(*
Nazwa:			P00_PneumaticValves
Opis:			Wyspa pneumatyczna
Wersja:			v1.0
Data:			2025-10-20
Autor:			DP
Urzadzenia:		Obsługa wyspy zaworowej
Konfiguracja:	
Info:
- kazdy zawór to 2 bity
#######################################################
#######################################################
*)



PROGRAM P00_PneumaticValves
VAR
	//ZMIENNE STERUJĄCE WYSPY ZAWOROWEJ
	QABPneumatic641ValveCoils 			AT %Q* 	: ARRAY[1..6] OF BYTE;
	QABPneumatic642ValveCoils 			AT %Q*	: ARRAY[1..5] OF BYTE;
	QABPneumatic643ValveCoils 			AT %Q*	: ARRAY[1..5] OF BYTE;
	QABPneumatic644ValveCoils 			AT %Q*	: ARRAY[1..5] OF BYTE;
	QABPneumatic645ValveCoils 			AT %Q*	: ARRAY[1..2] OF BYTE;
	QABPneumatic646ValveCoils 			AT %Q* 	: ARRAY[1..5] OF BYTE;
	QABPneumatic647ValveCoils 			AT %Q* 	: ARRAY[1..5] OF BYTE;
	QABPneumaticPI641ValveCoils 		AT %Q* 	: ARRAY[1..6] OF BYTE;

	QABPneumatic641PressureRegulator 	AT %Q* 	: ARRAY[1..2] OF BYTE;
	IABPneumatic641PressureRegulator 	AT %I* 	: ARRAY[1..2] OF BYTE;
	QABPneumatic645_1PressureRegulator 	AT %Q* 	: ARRAY[1..2] OF BYTE;
	IABPneumatic645_1PressureRegulator 	AT %I* 	: ARRAY[1..2] OF BYTE;
	QABPneumatic645_2PressureRegulator 	AT %Q* 	: ARRAY[1..2] OF BYTE;
	IABPneumatic645_2PressureRegulator 	AT %I* 	: ARRAY[1..2] OF BYTE;
	
	IABPneumatic641_N11AnalogInput1 	AT %I* 	: ARRAY[1..2] OF BYTE;
	IABPneumatic641_N11AnalogInput2 	AT %I* 	: ARRAY[1..2] OF BYTE;
	IABPneumatic641_N11AnalogInput3 	AT %I* 	: ARRAY[1..2] OF BYTE;
	IABPneumatic641_N11AnalogInput4 	AT %I* 	: ARRAY[1..2] OF BYTE;
	IABPneumatic645_N11AnalogInput1 	AT %I* 	: ARRAY[1..2] OF BYTE;
	IABPneumatic645_N11AnalogInput2 	AT %I* 	: ARRAY[1..2] OF BYTE;
	IABPneumatic645_N11AnalogInput3 	AT %I* 	: ARRAY[1..2] OF BYTE;
	IABPneumatic645_N11AnalogInput4 	AT %I* 	: ARRAY[1..2] OF BYTE;
	                                    
	IABPneumatic641_N12DigitalInput 	AT %I* 	: BYTE;	
	IABPneumatic642_N11DigitalInput 	AT %I* 	: BYTE;	
	IABPneumatic642_N12DigitalInput 	AT %I* 	: BYTE;	
	IABPneumatic642_N13DigitalInput 	AT %I* 	: BYTE;	
	IABPneumatic643_N11DigitalInput 	AT %I* 	: BYTE;	
	IABPneumatic643_N12DigitalInput 	AT %I* 	: BYTE;	
	IABPneumatic643_N13DigitalInput 	AT %I* 	: BYTE;
	IABPneumatic644_N11DigitalInput 	AT %I* 	: BYTE;	
	IABPneumatic644_N12DigitalInput 	AT %I* 	: BYTE;	
	IABPneumatic644_N13DigitalInput 	AT %I* 	: BYTE;
	IABPneumatic645_N12DigitalInput 	AT %I* 	: BYTE;
	IABPneumatic646_N11DigitalInput 	AT %I* 	: BYTE;
	IABPneumatic646_N12DigitalInput 	AT %I* 	: BYTE;
	IABPneumatic646_N13DigitalInput 	AT %I* 	: BYTE;
	IABPneumatic647_N11DigitalInput 	AT %I* 	: BYTE;
	IABPneumatic647_N12DigitalInput 	AT %I* 	: BYTE;
	IABPneumaticPI641_N11DigitalInput 	AT %I* 	: BYTE;
	IABPneumaticPI641_N12DigitalInput 	AT %I* 	: BYTE;
	IABPneumaticPI641_N13DigitalInput 	AT %I* 	: BYTE;
	                                  
	iIABPneumatic645_N11AnalogInput1	:INT;
	iIABPneumatic645_N11AnalogInput2    :INT;
	iIABPneumatic645_N11AnalogInput3    :INT;
	iIABPneumatic645_N11AnalogInput4    :INT;
	iIABPneumatic641_N11AnalogInput1    :INT;
	iIABPneumatic641_N11AnalogInput2    :INT;
	iIABPneumatic641_N11AnalogInput3    :INT;
	iIABPneumatic641_N11AnalogInput4    :INT;
	
	iIABPneumatic641PressureRegulator1				: INT;
	iIABPneumatic641PressureRegulator2				: INT;
	iIABPneumatic645_1PressureRegulator1			: INT;
	iIABPneumatic645_1PressureRegulator2			: INT;
	iIABPneumatic645_2PressureRegulator1			: INT;
	iIABPneumatic645_2PressureRegulator2			: INT;
	
	iQABPneumatic641PressureRegulator1				: INT;
	iQABPneumatic641PressureRegulator2				: INT;	
	iQABPneumatic645_1PressureRegulator1			: INT;
	iQABPneumatic645_1PressureRegulator2			: INT;
	iQABPneumatic645_2PressureRegulator1			: INT;
	iQABPneumatic645_2PressureRegulator2			: INT;	
	                                    
	(*Skalowanie czujników poziomu*)    
	fbiTank1LevelSensorValue 			: FB_4_20mA_TO_INT;
	fbiTank2LevelSensorValue 			: FB_4_20mA_TO_INT;	
	
	lrLidSealerPressureTemp						: LREAL;
	lrGripperScrewerCatchPressureTemp			: LREAL;
	lrGripperScrewerPressureTemp				: LREAL;
	lrDispencercatchPressureTemp				: LREAL;

	
END_VAR

//aVTEM();
//aVTEMSignals();
aAnalogueInput();
aDigitalInput();
aPressureRegulator();
aValveCoil();

ACTION aAnalogueInput:
(*
Nazwa:			aAnalogueInput
Opis:			Zawory pneumatyczne
Wersja:			v0.1
Data:			2024-10-28
Autor:			DP
Urzadzenia:		
Konfiguracja:	
Info:
- Czujnik pozycji Balluff, trzeba skonfigurować na 4-20mA, domyślnie jest na 0-10V
- Instrukcja konfiguracji czujnika: 2s, 1x, 1x (zniknie dioda), 2s (wyjście), 2s (wyjście)
*)

(*************************** 641N1.1 **************************************)
// Wyspa 1 - dozowanie
//AI1 4-20mA 
IABPneumatic641_N11AnalogInput1[1];
IABPneumatic641_N11AnalogInput1[2];
iIABPneumatic641_N11AnalogInput1	:= WORD_TO_INT(F_2Bytes_To_Word(byHigh:=IABPneumatic641_N11AnalogInput1[2],byLow:=IABPneumatic641_N11AnalogInput1[1]));
P02_Dispencers.IbDispencersCatch1SensorValue:=F_Scaling(rValue:=iIABPneumatic641_N11AnalogInput1, 
	rXmin:=		0,		//	0mA
	rXmax:=		32767,	//	23mA
	rYmin:= 	-70000, //	~10000 -> ~10mm (szyjka butelki) zamkniety (chwytak otwiera się na 49mm)
	rYmax:=		135000 );// ~60000 -> ~60mm otwarty
{warning 'dodać błąd czujnika poniżej 4mA i powyżej 20mA'}
IABPneumatic641_N11AnalogInput2[1]; 
IABPneumatic641_N11AnalogInput2[2];
iIABPneumatic641_N11AnalogInput2	:= WORD_TO_INT(F_2Bytes_To_Word(byHigh:=IABPneumatic641_N11AnalogInput2[2],byLow:=IABPneumatic641_N11AnalogInput2[1]));
P02_Dispencers.IbDispencersCatch2SensorValue:=F_Scaling(rValue:=iIABPneumatic641_N11AnalogInput2, 
	rXmin:=		0,		//	0mA
	rXmax:=		32767,	//	23mA
	rYmin:= 	-70000, //	~10000 -> ~10mm (szyjka butelki) zamkniety (chwytak otwiera się na 49mm)
	rYmax:=		135000 );// ~60000 -> ~60mm otwarty

IABPneumatic641_N11AnalogInput3[1]; 
IABPneumatic641_N11AnalogInput3[2]; 
iIABPneumatic641_N11AnalogInput3	:= WORD_TO_INT(F_2Bytes_To_Word(byHigh:=IABPneumatic641_N11AnalogInput3[2],byLow:=IABPneumatic641_N11AnalogInput3[1]));
P02_Dispencers.IbDispencersCatch3SensorValue:=F_Scaling(rValue:=iIABPneumatic641_N11AnalogInput3, 
	rXmin:=		0,		//	0mA
	rXmax:=		32767,	//	23mA
	rYmin:= 	-70000, //	~10000 -> ~10mm (szyjka butelki) zamkniety (chwytak otwiera się na 49mm)
	rYmax:=		135000 );// ~60000 -> ~60mm otwarty

IABPneumatic641_N11AnalogInput4[1]; 	
IABPneumatic641_N11AnalogInput4[2]; 
iIABPneumatic641_N11AnalogInput4	:= WORD_TO_INT(F_2Bytes_To_Word(byHigh:=IABPneumatic641_N11AnalogInput4[2],byLow:=IABPneumatic641_N11AnalogInput4[1]));
P02_Dispencers.IbDispencersCatch4SensorValue:=F_Scaling(rValue:=iIABPneumatic641_N11AnalogInput4, 
	rXmin:=		0,		//	0mA
	rXmax:=		32767,	//	23mA
	rYmin:= 	-70000, //	~10000 -> ~10mm (szyjka butelki) zamkniety (chwytak otwiera się na 49mm)
	rYmax:=		135000 );// ~60000 -> ~60mm otwarty

(*********************Koniec 641N1.1 **************************************)


(*************************** 645N1.1 **************************************)
// Wyspa 5 - zakręcarki i czujnik poziomu
//AI1 4-20mA 
IABPneumatic645_N11AnalogInput1[1];
IABPneumatic645_N11AnalogInput1[2];
iIABPneumatic645_N11AnalogInput1	:= WORD_TO_INT(F_2Bytes_To_Word(byHigh:=IABPneumatic645_N11AnalogInput1[2],byLow:=IABPneumatic645_N11AnalogInput1[1]));
P10_GripperScrewer.IlrGripperScrewer1HeightCV	:=	-0.0023*(iIABPneumatic645_N11AnalogInput1)+52.006 + 2.6788;

IABPneumatic645_N11AnalogInput2[1]; 
IABPneumatic645_N11AnalogInput2[2]; 
iIABPneumatic645_N11AnalogInput2	:= WORD_TO_INT(F_2Bytes_To_Word(byHigh:=IABPneumatic645_N11AnalogInput2[2],byLow:=IABPneumatic645_N11AnalogInput2[1]));
P10_GripperScrewer.IlrGripperScrewer2HeightCV	:=	-0.0023*(iIABPneumatic645_N11AnalogInput2)+52.006 + 2.252;

IABPneumatic645_N11AnalogInput3[1];
IABPneumatic645_N11AnalogInput3[2];
iIABPneumatic645_N11AnalogInput3	:= WORD_TO_INT(F_2Bytes_To_Word(byHigh:=IABPneumatic645_N11AnalogInput3[2],byLow:=IABPneumatic645_N11AnalogInput3[1]));
//iTank1Sensor1Value;//Czujnik poziomu 1
fbiTank1LevelSensorValue(
	iIN:= 	iIABPneumatic645_N11AnalogInput3, 
	rXmin:= 5190,//5513.0, 	// 4mA
	rXmax:= 27307.0, 	// 20mA
	rYmin:= 10.0, 		// 10mm na czujniku to 4mA
	rYmax:= 325.0,		// 325mm na czujniku to 20mA
	bError=>, 			// Bląd <4mA i >20mA
	iOUT=>	VIS.iTank1LevelSensorValue );
fbiTank1LevelSensorValue.bError;

IABPneumatic645_N11AnalogInput4[1];
IABPneumatic645_N11AnalogInput4[2];
iIABPneumatic645_N11AnalogInput4	:= WORD_TO_INT(F_2Bytes_To_Word(byHigh:=IABPneumatic645_N11AnalogInput4[2],byLow:=IABPneumatic645_N11AnalogInput4[1]));
//iTank2Sensor2Value;//Czujnik poziomu 2
fbiTank2LevelSensorValue(
	iIN:= 	iIABPneumatic645_N11AnalogInput4, 
	rXmin:= 5190,//5513.0, 	// 4mA
	rXmax:= 27307.0, 	// 20mA
	rYmin:= 10.0, 		// 10mm na czujniku to 4mA
	rYmax:= 325.0,		// 325mm na czujniku to 20mA
	bError=>, 			// Bląd <4mA i >20mA
	iOUT=>	VIS.iTank2LevelSensorValue );
fbiTank2LevelSensorValue.bError;
END_ACTION

ACTION aDigitalInput:
(*
Nazwa:			aDigitalInput
Opis:			Wejścia podłączone do wyspy pneumatycznej
Wersja:			v0.1
Data:			2024-10-28
Autor:			DP
Urzadzenia:		
Konfiguracja:	
Info:
*)
(* Stare z UBL50 Ziaja
(*************************** A3 **************************************)
// Wyspa 7 - podajnik opakowań
MAIN.IbLidSealerAfterSensor:=IABPneumaticA3DigitalInput[1].7;   //brak czujnika, póki co nie dokładamy
MAIN.IbBlowBeforeGripperScrewerSensor  :=	IABPneumaticA3DigitalInput[2].1;	  //czujnik pomiędzy UL a UF -> (opcja) być moze do usunięcia
MAIN.IbCapSorterFirstFormCheckFormSensor := IABPneumaticA3DigitalInput[2].2;	
MAIN.IbCapSorterAfterFormSensor2 :=	IABPneumaticA3DigitalInput[2].3;	//Czujnik drag sortera nakretek	

*)

(*************************** 641N1.2 **************************************)
P02_Dispencers.IbDispencer1DropCatcherBackSensor		:=	IABPneumatic641_N12DigitalInput.0;
P02_Dispencers.IbDispencer2DropCatcherBackSensor		:=	IABPneumatic641_N12DigitalInput.1;
P02_Dispencers.IbDispencer3DropCatcherBackSensor		:=	IABPneumatic641_N12DigitalInput.2;
P02_Dispencers.IbDispencer4DropCatcherBackSensor		:=	IABPneumatic641_N12DigitalInput.3;
P01_BottleFeeder.IbBottleFeederNotInsertedSensor		:=	IABPneumatic641_N12DigitalInput.4;
GVL_IO.IbPressureInSystemSensor							:=  IABPneumatic641_N12DigitalInput.5; //ciśnienie robocze ok za zaworem bezpieczęństwa? 
P02_Dispencers.IbDispencer12NoColisionWhenDosingSensor	:=	IABPneumatic641_N12DigitalInput.6; //rezerwa
P02_Dispencers.IbDispencer34NoColisionWhenDosingSensor	:=	IABPneumatic641_N12DigitalInput.7; //rezerwa

(*************************** 642N1.1 **************************************)
P16_LabelMachine.IbLabelMachineFullSensor			:=	IABPneumatic642_N11DigitalInput.0;
P14_BadBottleConyevor.IbBadBottleConveyorFullSensor	:=	IABPneumatic642_N11DigitalInput.1;
MAIN.IbBottleInFormCheckBottleSensor				:=	IABPneumatic642_N11DigitalInput.2;
P13_BottleTransfer.IbBottleCheckAfterBottleTransferSensor	:=	IABPneumatic642_N11DigitalInput.3;
MAIN.IbFormCheckFormSensor							:=	IABPneumatic642_N11DigitalInput.4;
MAIN.IbFourthFormCheckFormSensor					:=	IABPneumatic642_N11DigitalInput.5;
MAIN.IbSecondFormCheckFormSensor			:=	IABPneumatic642_N11DigitalInput.6;	
P02_Dispencers.IbDispencerAfterCheckFormSensor		:=	IABPneumatic642_N11DigitalInput.7;

(*************************** 642N1.2 **************************************)
P13_BottleTransfer.IbFirstFormCheckFormSensor		:=	IABPneumatic642_N12DigitalInput.0;
P13_BottleTransfer.IbSecondFormCheckFormSensor	:=	IABPneumatic642_N12DigitalInput.1;
P13_BottleTransfer.IbBottleTransferFormAfterSensor	:=	IABPneumatic642_N12DigitalInput.2;
P13_BottleTransfer.IbBottleTransferFormAfterSensor2	:=	IABPneumatic642_N12DigitalInput.3;	//czujnik nr 2 kolejki za robotem ?
P01_TwoPhasesBarriers.IbBarrierBetweenDispencerOpenedSensor	:=	IABPneumatic642_N12DigitalInput.4;
P01_TwoPhasesBarriers.IbBarrierBetweenDispencerClosedSensor	:=	IABPneumatic642_N12DigitalInput.5;
P01_TwoPhasesBarriers.IbBarrierBetweenWeightOpenedSensor	:=	IABPneumatic642_N12DigitalInput.6;
P01_TwoPhasesBarriers.IbBarrierBetweenWeightClosedSensor	:=	IABPneumatic642_N12DigitalInput.7;

(*************************** 642N1.3 **************************************)
P02_Dispencers.IbDispencersDragLeftDragUpSensor			:=	IABPneumatic642_N13DigitalInput.0;
P02_Dispencers.IbDispencersDragLeftDragDownSensor		:=	IABPneumatic642_N13DigitalInput.1;
P02_Dispencers.IbDispencersDragLeftDragHomingSensor		:=	IABPneumatic642_N13DigitalInput.2;
P02_Dispencers.IbDispencersDragRightDragUpSensor		:=	IABPneumatic642_N13DigitalInput.3;
P02_Dispencers.IbDispencersDragRightDragDownSensor		:=	IABPneumatic642_N13DigitalInput.4;
P02_Dispencers.IbDispencersDragRightDragHomingSensor	:=	IABPneumatic642_N13DigitalInput.5;
P02_Dispencers.IbDispencersDragLeftLeadBefore1UpSensor	:=	IABPneumatic642_N13DigitalInput.6;
P02_Dispencers.IbDispencersDragRightLeadBefore1UpSensor	:=	IABPneumatic642_N13DigitalInput.7;

(*************************** 643N1.1 **************************************)
MAIN.IbTwoPhasesFormSensorBetweenDispencers		:=	IABPneumatic643_N11DigitalInput.0;
P01_Gates.IbGateBeforeWeights14Sensor			:=	IABPneumatic643_N11DigitalInput.1;							//obecność formatki przy rfid za 1 faza dozowniki
P01_Gates.IbGateBeforeWeights56Sensor			:=	IABPneumatic643_N11DigitalInput.2;							//obecność formatki przy rfid za 2 faza dozowniki
P05_Weight.IbWeight1FormSensor					:=	IABPneumatic643_N11DigitalInput.3;
P05_Weight.IbWeight2FormSensor					:=	IABPneumatic643_N11DigitalInput.4;
P05_Weight.IbWeight3FormSensor					:=	IABPneumatic643_N11DigitalInput.5;
P05_Weight.IbWeight4FormSensor					:=	IABPneumatic643_N11DigitalInput.6;
P06_LidFeeder.IbLidFeederFirstFormSensorBeforeDrag	:=	IABPneumatic643_N11DigitalInput.7;								//obecność 1 formatki przed podawaniem platynek
;
(*************************** 643N1.2 **************************************)
MAIN.IbLidFeederThirdFormSensor	:=	IABPneumatic643_N12DigitalInput.0;									//obecność 2 formatki przed podawaniem platynek
MAIN.IbLidFeederAfterSensor	:=	IABPneumatic643_N12DigitalInput.1;									//obecność formatki przy rfid przed przygrzewaniem platynek
P11_CapCorrectCheck.IbCapCorrectCheckAfterScrewerFormSensor	:=	IABPneumatic643_N12DigitalInput.2;		//kolejka formatek za zakręcarkami
P11_CapCorrectCheck.IbCapCorrectCheckFormSensor	:=	IABPneumatic643_N12DigitalInput.3;									//obecność formatki przy rfid kontrola zamknięcia	
P11_CapCorrectCheck.IbCapCorrectCheckBottleSensor	:=	IABPneumatic643_N12DigitalInput.4;		
P05_Weight.IbWeight6FormSensor :=	IABPneumatic643_N12DigitalInput.5;									
P05_Weight.IbWeight5FormSensor :=	IABPneumatic643_N12DigitalInput.6;									
IABPneumatic643_N12DigitalInput.7;										//rezerwa

(*************************** 643N1.3 **************************************)
IABPneumatic643_N13DigitalInput.0;	//szlaban przed wagami 1-4
P01_TwoPhasesBarriers.IbGateBeforeWeights56		:=	IABPneumatic643_N13DigitalInput.1;
P02_Dispencers.IbDispencersDragLeftLeadAfter1UpSensor		:=	IABPneumatic643_N13DigitalInput.2;
P02_Dispencers.IbDispencersDragRightLeadAfter1UpSensor		:=	IABPneumatic643_N13DigitalInput.3;
MAIN.IbLidSealerFirstFormSensor		:=	IABPneumatic643_N13DigitalInput.4;		// Czujnik obecności 1-ej formatki przygrzewacze platynek
MAIN.IbLidSealerSecondFormSensor	:=	IABPneumatic643_N13DigitalInput.5;	// Czujnik obecności 2-ej formatki przygrzewacze platynek 
IABPneumatic643_N13DigitalInput.6;	//rezerwa
IABPneumatic643_N13DigitalInput.7;	//rezerwa

(*************************** 644N1.1 **************************************)
MAIN.IbLidSealerAfterSensor	:=	IABPneumatic644_N11DigitalInput.0;									//czujnik formatki za przygrzewaczami
P10_GripperScrewer.IbGripperScrewersSixthFormCheckFormSensor		:=	IABPneumatic644_N11DigitalInput.1;	
P09_CapPuttedCheck.IbCapPuttedCheckFormSensor	:=	IABPneumatic644_N11DigitalInput.2;									//obecność formatki przy rfid przed zakręcarkami
P10_GripperScrewer.IbGripperScrewersBeforeThirdFormCheckFormSensor 	:=	IABPneumatic644_N11DigitalInput.3;
P10_GripperScrewer.IbGripperScrewersThirdFormCheckFormSensor		:=	IABPneumatic644_N11DigitalInput.4;
P11_CapCorrectCheck.IbCapCorrectCheckDialAfterScrewerFormSensor		:=	IABPneumatic644_N11DigitalInput.5;
P01_Gates.IbLidFeederBarrierOnSensor								:=	IABPneumatic644_N11DigitalInput.6;	//banda opuszczona pomiędzy podawaniem a przygrzewaniem platynek
P01_Gates.IbLidFeederBarrierOffSensor								:=	IABPneumatic644_N11DigitalInput.7;	//banda podniesiona pomiędzy podawaniem a przygrzewaniem platynek

(*************************** 644N1.2 **************************************)
//Platynki
(*P06_LidFeeder.IbLidFeederFormPositioning1HideSensor	:=	IABPneumatic644_N12DigitalInput.0;	//pozycjonowanie formatki pod podajnikiem platynek wsynięte
P06_LidFeeder.IbLidFeederFormPositioning2HideSensor	:=	IABPneumatic644_N12DigitalInput.1;	//pozycjonowanie formatki pod podajnikiem platynek wysunięte
P06_LidFeeder.IbLidFeederDragLeadBefore1UpSensor	:=	NOT IABPneumatic644_N12DigitalInput.2;
P06_LidFeeder.IbLidFeederDragUpSensor				:=	IABPneumatic644_N12DigitalInput.3;
P06_LidFeeder.IbLidFeederDragDownSensor				:=	IABPneumatic644_N12DigitalInput.4;
P06_LidFeeder.IbLidFeederDragHomingSensor			:=	IABPneumatic644_N12DigitalInput.5;
P06_LidSealer.IbLidSealerDragLeadBefore1UpSensor	:=	NOT IABPneumatic644_N12DigitalInput.6;
P06_LidSealer.IbLidSealerDragUpSensor				:=	IABPneumatic644_N12DigitalInput.7;*)
//Podajnik knotów
P06_WickFeeder.IbFormPositioningHide1				:=	IABPneumatic644_N12DigitalInput.0;	//pozycjonowanie formatki pod podajnikiem platynek wsynięte
P06_WickFeeder.IbFormPositioningHide2				:=	IABPneumatic644_N12DigitalInput.1;	//pozycjonowanie formatki pod podajnikiem platynek wysunięte
P06_WickFeeder.IbWickFeederDragLeadBefore1UpSensor	:=	IABPneumatic644_N12DigitalInput.2;
P06_WickFeeder.IbWickFeederDragUpSensor				:=	IABPneumatic644_N12DigitalInput.3;
P06_WickFeeder.IbWickFeederDragDownSensor			:=	IABPneumatic644_N12DigitalInput.4;
P06_WickFeeder.IbWickFeederDragHomingSensor			:=	IABPneumatic644_N12DigitalInput.5;
P06_LidSealer.IbLidSealerDragLeadBefore1UpSensor	:=	IABPneumatic644_N12DigitalInput.6;
P06_LidSealer.IbLidSealerDragUpSensor				:=	IABPneumatic644_N12DigitalInput.7;
(*************************** 644N1.3 **************************************)
P06_LidSealer.IbLidSealerDragDownSensor						:=	IABPneumatic644_N13DigitalInput.0;
P06_LidSealer.IbLidSealerDragHomingSensor					:=	IABPneumatic644_N13DigitalInput.1;
P10_GripperScrewer.IbGripperScrewersDragLeadBefore1UpSensor	:=	IABPneumatic644_N13DigitalInput.2;
P10_GripperScrewer.IbGripperScrewersDragLeadBefore2UpSensor	:=	IABPneumatic644_N13DigitalInput.3;
P10_GripperScrewer.IbGripperScrewersDragUpSensor			:=	IABPneumatic644_N13DigitalInput.4;
P10_GripperScrewer.IbGripperScrewersDragDownSensor			:=	IABPneumatic644_N13DigitalInput.5;
P10_GripperScrewer.IbGripperScrewersDragHomingSensor		:=	IABPneumatic644_N13DigitalInput.6;
IABPneumatic644_N13DigitalInput.7;	//rezerwa

(*************************** 645N1.2 **************************************)
P09_CapPuttedCheck.IbCapPuttedCheckSensor					:=	IABPneumatic645_N12DigitalInput.0;
P11_CapCorrectCheck.IbCapCorrectCheckCapOKSensor			:=	IABPneumatic645_N12DigitalInput.1;
P11_CapCorrectCheck.IbCapCorrectCheckCapNotScrewedSensor	:=	IABPneumatic645_N12DigitalInput.2;
IABPneumatic645_N12DigitalInput.3;	//chwytak zakręcarki otwarty				//brak fizycznie !!
IABPneumatic645_N12DigitalInput.4;	//chwytak zakręcarki zamknięty              //brak fizycznie !!
IABPneumatic645_N12DigitalInput.5;	//rezerwa
IABPneumatic645_N12DigitalInput.6;	//rezerwa
IABPneumatic645_N12DigitalInput.7;	//rezerwa

(*************************** 646N1.1 **************************************)
//Platynki
(*P06_LidFeeder.IbLidFeederUpSensor2		:=	IABPneumatic646_N11DigitalInput.0;	//głowica wieczek 1 u góry
P06_LidFeeder.IbLidFeederDownSensor2	:=	IABPneumatic646_N11DigitalInput.1;  //głowica wieczek 1 w dole
P06_LidFeeder.IbLidFeederUpSensor1		:=	IABPneumatic646_N11DigitalInput.2;  //głowica wieczek 2 u góry
P06_LidFeeder.IbLidFeederDownSensor1	:=	IABPneumatic646_N11DigitalInput.3;  //głowica wieczek 2 w dole
P06_LidFeeder.IbLidFeederLowLevelSensor2 :=	NOT IABPneumatic646_N11DigitalInput.4;  //obecność wieczek zbiornik 1
P06_LidFeeder.IbLidFeederLowLevelSensor1 :=	NOT IABPneumatic646_N11DigitalInput.5;  //obecność wieczek zbiornik 2
P06_LidFeeder.IbLidFeeder2SuckerSensor			:= IABPneumatic646_N11DigitalInput.6;  //rezerwa    //podciśnienie podsysania wieczka OK
P06_LidFeeder.IbLidFeederSuckerSensor	:=	IABPneumatic646_N11DigitalInput.7;  //rezerwa	//podciśnienie podsysania wieczka OK

IABPneumatic646_N12DigitalInput.0;	//rezerwa
IABPneumatic646_N12DigitalInput.1;  //rezerwa
IABPneumatic646_N12DigitalInput.2;  //rezerwa
IABPneumatic646_N12DigitalInput.3;  //rezerwa
IABPneumatic646_N12DigitalInput.4;  //rezerwa
IABPneumatic646_N12DigitalInput.5;  //rezerwa
IABPneumatic646_N12DigitalInput.6;  //rezerwa
IABPneumatic646_N12DigitalInput.7;  //rezerwa*)
//Knoty
P06_WickFeeder.IbQueFullSensor															:=	IABPneumatic646_N11DigitalInput.0;	
P06_WickFeeder.IbWheelSensor															:=	IABPneumatic646_N11DigitalInput.1; 
P06_WickFeeder.IbWheelLevelSensor														:=	IABPneumatic646_N11DigitalInput.2;  
P06_WickFeeder.IbWickAtPipe																:=	IABPneumatic646_N11DigitalInput.3;  
P06_WickFeeder.IbSeparatorPos1															:=	IABPneumatic646_N11DigitalInput.4;  
P06_WickFeeder.IbSeparatorPos2															:=		IABPneumatic646_N11DigitalInput.5;  
P06_WickFeeder.IbSleve1SeparatorOut														:= IABPneumatic646_N11DigitalInput.6; 
P06_WickFeeder.IbQueFullAtSleve1														:=	IABPneumatic646_N11DigitalInput.7; 

P06_WickFeeder.IbSleve2SeparatorOut														:=	IABPneumatic646_N12DigitalInput.0;	
P06_WickFeeder.IbQueFullAtSleve2														:=	IABPneumatic646_N12DigitalInput.1;  
P06_WickFeeder.IbWickAtSleve1															:=	IABPneumatic646_N12DigitalInput.2;  
P06_WickFeeder.IbWickAtSleve2															:=	IABPneumatic646_N12DigitalInput.3;  
P06_WickFeeder.IbHammer1Down															:=	IABPneumatic646_N12DigitalInput.4;  
P06_WickFeeder.IbHammer1Up																:=	IABPneumatic646_N12DigitalInput.5;  
P06_WickFeeder.IbHammer2Down															:=	IABPneumatic646_N12DigitalInput.6;  
P06_WickFeeder.IbHammer2Up																:=	IABPneumatic646_N12DigitalInput.7;  

P06_WickFeeder.IbQueFullAfterWheelSensor 												:=	IABPneumatic646_N13DigitalInput.0;	
IABPneumatic646_N13DigitalInput.1;  
IABPneumatic646_N13DigitalInput.2;  
IABPneumatic646_N13DigitalInput.3;  
IABPneumatic646_N13DigitalInput.4;  
IABPneumatic646_N13DigitalInput.5;  
IABPneumatic646_N13DigitalInput.6;  
IABPneumatic646_N13DigitalInput.7;  


(*************************** A3 **************************************)
// Wyspa 7 - podajnik opakowań
//DI1
P08_CapSorter.IbCapSorterDragUpSensor:=  IABPneumatic647_N11DigitalInput.0;	// widły pod podajnikiem zamknięć wysunięte
P08_CapSorter.IbCapSorterDragDownSensor:=  IABPneumatic647_N11DigitalInput.1;	 //widły pod podajnikiem zamknięć schowane
P08_CapSorter.IbCapSorterDragHomingSensor:= IABPneumatic647_N11DigitalInput.2;	//prowadzenie formatek przed podajnikiem zamknięć lewe podniesione
P08_CapSorter.IbCapSorterDragLeadBefore1UpSensor:=  IABPneumatic647_N11DigitalInput.3;	//prowadzenie formatek przed podajnikiem zamknięć lewe podniesione
P08_CapSorter.IbCapSorterDragLeadBefore2UpSensor:=  IABPneumatic647_N11DigitalInput.4;	//prowadzenie formatek przed podajnikiem zamknięć prawe podniesione
P08_CapSorter.IbCapSorterDragLeadAfter1UpSensor:=IABPneumatic647_N11DigitalInput.5;	//czujnik wjazdu przed podajnikiem zamknięć 
P08_CapSorter.IbCapSorterDragLeadAfter2UpSensor:=IABPneumatic647_N11DigitalInput.6;	// czujnik  4 formatki za podajnikiem zamknięć -> czujnik na ukos
;IABPneumatic647_N11DigitalInput.7;   //brak czujnika, póki co nie dokładamy
//DI2
MAIN.IbCapSorterFirstFormCheckFormSensor := IABPneumatic647_N12DigitalInput.0;	   //ostatnia formatka przed przeciąganiem
MAIN.IbCapSorterAfterFormSensor2  :=	IABPneumatic647_N12DigitalInput.1;	  //czujnik pomiędzy UL a UF -> (opcja) być moze do usunięcia
MAIN.IbCapSorterBeforeFourthFormCheckFormSensor := IABPneumatic647_N12DigitalInput.2;	
MAIN.IbCapSorterFourthFormCheckFormSensor :=	IABPneumatic647_N12DigitalInput.3;	//Czujnik drag sortera nakretek
MAIN.IbBlowBeforeGripperScrewerSensor := IABPneumatic647_N12DigitalInput.4;	
MAIN.IbCapSorterAfterFormSensor := IABPneumatic647_N12DigitalInput.5;		
IABPneumatic647_N12DigitalInput.6;		
IABPneumatic647_N12DigitalInput.7;		

(*********************Koniec A3 **************************************)

(*************************** 641**************************************)
// Wyspa 6 - podajnik opakowań
P01_pucksInserter.IbPucksInserterLevelSensor				:= IABPneumaticPI641_N11DigitalInput.0;	
P01_pucksInserter.IbPucksInserterWheelEntrySensor			:= IABPneumaticPI641_N11DigitalInput.1;	
P01_pucksInserter.IbPucksInserterWheelExitSensor			:= IABPneumaticPI641_N11DigitalInput.2;	
P01_pucksInserter.IbPucksInserterFormGateBeforeSensor		:= IABPneumaticPI641_N11DigitalInput.3;	
P01_pucksInserter.IbPucksInserterFormGateAfterSensor		:= IABPneumaticPI641_N11DigitalInput.4;	//czujnik kolejki Stołu podającego
P01_pucksInserter.IbPucksInserterHammerUpSensor				:= IABPneumaticPI641_N11DigitalInput.5;		
P01_pucksInserter.IbPucksInserterHammerDownSensor			:= IABPneumaticPI641_N11DigitalInput.6;		
P01_pucksInserter.IbPucksInserterTrayOffSensor				:= IABPneumaticPI641_N11DigitalInput.7;	
//DI2
P01_pucksInserter.IbPucksInserterTrayOnSensor				:= IABPneumaticPI641_N12DigitalInput.0;	
P01_pucksInserter.IbPucksInserterFormPositioningOffSensor	:= IABPneumaticPI641_N12DigitalInput.1;	
P01_pucksInserter.IbPucksInserterFormPositioningOnSensor	:= IABPneumaticPI641_N12DigitalInput.2;	
P01_pucksInserter.IbPucksInserterGate1OffSensor				:= IABPneumaticPI641_N12DigitalInput.3;	
P01_pucksInserter.IbPucksInserterGate1OnSensor				:= IABPneumaticPI641_N12DigitalInput.4;	
P01_pucksInserter.IbPucksInserterGate2OffSensor				:= IABPneumaticPI641_N12DigitalInput.5;
P01_pucksInserter.IbPucksInserterGate2OnSensor				:= IABPneumaticPI641_N12DigitalInput.6;		
P01_pucksInserter.IbPucksInserterHomingSensor				:= IABPneumaticPI641_N12DigitalInput.7;	

 P01_pucksInserter.IbPucksInserterPushTablesSensor			:= IABPneumaticPI641_N13DigitalInput.0;	
 IABPneumaticPI641_N13DigitalInput.1;	
 IABPneumaticPI641_N13DigitalInput.2;	
 IABPneumaticPI641_N13DigitalInput.3;	
 IABPneumaticPI641_N13DigitalInput.4;	
 IABPneumaticPI641_N13DigitalInput.5;
 IABPneumaticPI641_N13DigitalInput.6;	
 IABPneumaticPI641_N13DigitalInput.7;	



(*********************Koniec 641 **************************************)
END_ACTION

ACTION aPressureRegulator:
(*
Nazwa:			aPressureRegulator
Opis:			Zawory pneumatyczne
Wersja:			v1.0
Data:			2025-10-20
Autor:			DP
Urzadzenia:		
Konfiguracja:	
Info:
*)
IF VIS.lrDispencerCatchPressureShow <3.5 THEN
	VIS.lrDispencerCatchPressureShow  :=5;
END_IF
IF VIS.lrDispencerCatchPressureShow >12 THEN
	VIS.lrDispencerCatchPressureShow  :=12;
END_IF

lrDispencercatchPressureTemp := ((lrDispencerCatchPressure*10)/14.8)*1000;
lrGripperScrewerCatchPressureTemp := ((lrGripperScrewerCatchPressure*10)/26.2)*1000;
lrGripperScrewerPressureTemp := ((lrGripperScrewerPressure*10)/14.8)*1000;

iQABPneumatic641PressureRegulator1 := LREAL_TO_INT(lrDispencercatchPressureTemp);
iQABPneumatic645_1PressureRegulator1 := LREAL_TO_INT(lrGripperScrewerCatchPressureTemp);
iQABPneumatic645_2PressureRegulator2 := LREAL_TO_INT(lrGripperScrewerPressureTemp);
	
(*************************** 641 **************************************)
// Wyspa 1 - dozowanie
QABPneumatic641PressureRegulator[1].0		:= iQABPneumatic641PressureRegulator1.0; 
QABPneumatic641PressureRegulator[1].1		:= iQABPneumatic641PressureRegulator1.1;                 
QABPneumatic641PressureRegulator[1].2		:= iQABPneumatic641PressureRegulator1.2;
QABPneumatic641PressureRegulator[1].3		:= iQABPneumatic641PressureRegulator1.3;
QABPneumatic641PressureRegulator[1].4		:= iQABPneumatic641PressureRegulator1.4;
QABPneumatic641PressureRegulator[1].5		:= iQABPneumatic641PressureRegulator1.5;
QABPneumatic641PressureRegulator[1].6		:= iQABPneumatic641PressureRegulator1.6;
QABPneumatic641PressureRegulator[1].7		:= iQABPneumatic641PressureRegulator1.7;
QABPneumatic641PressureRegulator[2].0		:= iQABPneumatic641PressureRegulator1.8; 
QABPneumatic641PressureRegulator[2].1		:= iQABPneumatic641PressureRegulator1.9;                 
QABPneumatic641PressureRegulator[2].2		:= iQABPneumatic641PressureRegulator1.10;
QABPneumatic641PressureRegulator[2].3		:= iQABPneumatic641PressureRegulator1.11;
QABPneumatic641PressureRegulator[2].4		:= iQABPneumatic641PressureRegulator1.12;
QABPneumatic641PressureRegulator[2].5		:= iQABPneumatic641PressureRegulator1.13;
QABPneumatic641PressureRegulator[2].6		:= iQABPneumatic641PressureRegulator1.14;
QABPneumatic641PressureRegulator[2].7		:= iQABPneumatic641PressureRegulator1.15;

IABPneumatic641PressureRegulator[1];
IABPneumatic641PressureRegulator[2];
iIABPneumatic641PressureRegulator1	:= WORD_TO_INT(F_2Bytes_To_Word(byHigh:=IABPneumatic641PressureRegulator[2],byLow:=IABPneumatic641PressureRegulator[1]));

(*********************Koniec 641 **************************************)

(*************************** 645 **************************************)
// Wyspa 5 - zakręcarki

//PR1
QABPneumatic645_1PressureRegulator[1];
QABPneumatic645_1PressureRegulator[2];
//Zawór proporcjonalny chwytaki pod zakręcarkami szczękowymi
QABPneumatic645_1PressureRegulator[1].0		:= iQABPneumatic645_1PressureRegulator1.0; 
QABPneumatic645_1PressureRegulator[1].1		:= iQABPneumatic645_1PressureRegulator1.1;                 
QABPneumatic645_1PressureRegulator[1].2		:= iQABPneumatic645_1PressureRegulator1.2;
QABPneumatic645_1PressureRegulator[1].3		:= iQABPneumatic645_1PressureRegulator1.3;
QABPneumatic645_1PressureRegulator[1].4		:= iQABPneumatic645_1PressureRegulator1.4;
QABPneumatic645_1PressureRegulator[1].5		:= iQABPneumatic645_1PressureRegulator1.5;
QABPneumatic645_1PressureRegulator[1].6		:= iQABPneumatic645_1PressureRegulator1.6;
QABPneumatic645_1PressureRegulator[1].7		:= iQABPneumatic645_1PressureRegulator1.7;
QABPneumatic645_1PressureRegulator[2].0		:= iQABPneumatic645_1PressureRegulator1.8; 
QABPneumatic645_1PressureRegulator[2].1		:= iQABPneumatic645_1PressureRegulator1.9;                 
QABPneumatic645_1PressureRegulator[2].2		:= iQABPneumatic645_1PressureRegulator1.10;
QABPneumatic645_1PressureRegulator[2].3		:= iQABPneumatic645_1PressureRegulator1.11;
QABPneumatic645_1PressureRegulator[2].4		:= iQABPneumatic645_1PressureRegulator1.12;
QABPneumatic645_1PressureRegulator[2].5		:= iQABPneumatic645_1PressureRegulator1.13;
QABPneumatic645_1PressureRegulator[2].6		:= iQABPneumatic645_1PressureRegulator1.14;
QABPneumatic645_1PressureRegulator[2].7		:= iQABPneumatic645_1PressureRegulator1.15;

IABPneumatic645_1PressureRegulator[1];
IABPneumatic645_1PressureRegulator[2];
iIABPneumatic645_1PressureRegulator1	:= WORD_TO_INT(F_2Bytes_To_Word(byHigh:=IABPneumatic645_1PressureRegulator[2],byLow:=IABPneumatic645_1PressureRegulator[1]));
 

//Zawór proporcjonalny chwytaki pod zakręcarkami szczękowymi
QABPneumatic645_2PressureRegulator[1].0		:= iQABPneumatic645_2PressureRegulator2.0; 
QABPneumatic645_2PressureRegulator[1].1		:= iQABPneumatic645_2PressureRegulator2.1;                 
QABPneumatic645_2PressureRegulator[1].2		:= iQABPneumatic645_2PressureRegulator2.2;
QABPneumatic645_2PressureRegulator[1].3		:= iQABPneumatic645_2PressureRegulator2.3;
QABPneumatic645_2PressureRegulator[1].4		:= iQABPneumatic645_2PressureRegulator2.4;
QABPneumatic645_2PressureRegulator[1].5		:= iQABPneumatic645_2PressureRegulator2.5;
QABPneumatic645_2PressureRegulator[1].6		:= iQABPneumatic645_2PressureRegulator2.6;
QABPneumatic645_2PressureRegulator[1].7		:= iQABPneumatic645_2PressureRegulator2.7;
QABPneumatic645_2PressureRegulator[2].0		:= iQABPneumatic645_2PressureRegulator2.8; 
QABPneumatic645_2PressureRegulator[2].1		:= iQABPneumatic645_2PressureRegulator2.9;                 
QABPneumatic645_2PressureRegulator[2].2		:= iQABPneumatic645_2PressureRegulator2.10;
QABPneumatic645_2PressureRegulator[2].3		:= iQABPneumatic645_2PressureRegulator2.11;
QABPneumatic645_2PressureRegulator[2].4		:= iQABPneumatic645_2PressureRegulator2.12;
QABPneumatic645_2PressureRegulator[2].5		:= iQABPneumatic645_2PressureRegulator2.13;
QABPneumatic645_2PressureRegulator[2].6		:= iQABPneumatic645_2PressureRegulator2.14;
QABPneumatic645_2PressureRegulator[2].7		:= iQABPneumatic645_2PressureRegulator2.15;
                           
IABPneumatic645_2PressureRegulator[1];
IABPneumatic645_2PressureRegulator[2];
iIABPneumatic645_2PressureRegulator1	:= WORD_TO_INT(F_2Bytes_To_Word(byHigh:=IABPneumatic645_2PressureRegulator[2],byLow:=IABPneumatic645_2PressureRegulator[1]));

(*********************Koniec 645 **************************************)
END_ACTION

ACTION aValveCoil:
(*
Nazwa:			aValveCoil
Opis:			Zawory pneumatyczne
Wersja:			v0.1
Data:			2024-10-28
Autor:			DP
Urzadzenia:		
Konfiguracja:	
Info:
*)

//Do podpięcia
P01_TwoPhasesBarriers.QbBarrierBetweenDispencerActuator;	
P01_TwoPhasesBarriers.QbBarrierBetweenWeightActuator;
P01_Gates.QbGate0BeforeDispencersActuator;
P01_Gates.QbGateBeforeDispencersActuator;
P01_Gates.QbLidFeederBarrierActuator;
P01_Gates.QbGateBeforeWeight14Actuator;
P01_Gates.QbGateBeforeWeight56Actuator;
P01_Gates.QbBottleTransferGate1Actuator;
 
P01_BottleFeeder.QbBottleFeederGate1;			
P01_BottleFeeder.QbBottleFeederGate2;					
P01_BottleFeeder.QbBottleFeederArmLeft;			
P01_BottleFeeder.QbBottleFeederArmDown;			
P01_BottleFeeder.QbBottleFeederGripper;			
P01_BottleFeeder.QbBottleFeederFormPositioning;	
P01_BottleFeeder.QbBottleFeederFormGate;			

P01_PucksInserter.QbPucksInserterHammer;
P01_PucksInserter.QbPucksInserterTray;
P01_PucksInserter.QbPucksInserterGate1;
P01_PucksInserter.QbPucksInserterGate2;
P01_PucksInserter.QbPucksInserterFormGate;
P01_PucksInserter.QbPucksInserterFormPositioning;

P02_Dispencers.QbDispencersDragRightDragActuator;
P02_Dispencers.QbDispencersDragLeftDragActuator;
P02_Dispencers.QbDispencersDragLeftLeadBefore1Actuator;
P02_Dispencers.QbDispencersDragLeftLeadAfter1Actuator;
P02_Dispencers.QbDispencersDragRightLeadBefore1Actuator;
P02_Dispencers.QbDispencersDragRightLeadAfter1Actuator;

P02_Dispencers.QbDispencer1SuckingValveActuator;
P02_Dispencers.QbDispencer2SuckingValveActuator;
P02_Dispencers.QbDispencer3SuckingValveActuator;
P02_Dispencers.QbDispencer4SuckingValveActuator;
P02_Dispencers.QbDispencer1DosingValveActuator;
P02_Dispencers.QbDispencer2DosingValveActuator;
P02_Dispencers.QbDispencer3DosingValveActuator;
P02_Dispencers.QbDispencer4DosingValveActuator;
P02_Dispencers.QbDispencersCatch1Actuator;
P02_Dispencers.QbDispencersCatch2Actuator;
P02_Dispencers.QbDispencersCatch3Actuator;
P02_Dispencers.QbDispencersCatch4Actuator;
P02_Dispencers.QbDispencer1DropCatcherValveActuator;
P02_Dispencers.QbDispencer2DropCatcherValveActuator;
P02_Dispencers.QbDispencer3DropCatcherValveActuator;
P02_Dispencers.QbDispencer4DropCatcherValveActuator;
P02_Dispencers.QbDispencersCatchMaxPressure;
P02_Dispencers.QbTank1Pressure;
P02_Dispencers.QbDispencerDropCatcherSuck;

P05_Weight.QbWeight1Actuator;
P05_Weight.QbWeight2Actuator;
P05_Weight.QbWeight3Actuator;
P05_Weight.QbWeight4Actuator;
P05_Weight.QbWeight5Actuator;
P05_Weight.QbWeight6Actuator;

P06_LidFeeder.QbLidFeederDragActuator;
P06_LidFeeder.QbLidFeederDragLeadBefore1Actuator;

P06_LidFeeder.QbLidFeeder_FeederActuator1;
P06_LidFeeder.QbLidFeeder_FeederActuator2;
P06_LidFeeder.QbLidFeeder2_FeederActuator1;
P06_LidFeeder.QbLidFeeder2_FeederActuator2;
P06_LidFeeder.QbLidFeeder2_HeaterActuator;
P06_LidFeeder.QbLidFeeder_HeaterActuator;
P06_LidFeeder.QbLidFeederBlockActuator;
P06_LidFeeder.QbLidFeederFormPositioningActuator; 

P06_LidSealer.QbLidSealer_SealingActuator;
P06_LidSealer.QbLidSealer2_SealingActuator;
P06_LidSealer.QbLidSealerDragActuator;
P06_LidSealer.QbLidSealerBlockActuator;
P06_LidSealer.QbLidSealerDragLeadBefore1Actuator;

P08_CapSorter.QbCapSorterDragActuator;
P08_CapSorter.QbCapSorterDragLeadBefore1Actuator;
P08_CapSorter.QbCapSorterStoperActuator;
QbBlowBeforeGripperScrewer;

QbGateBeforeGripperScrewer;
P10_GripperScrewer.QbGripperScrewersDragActuator;
P10_GripperScrewer.QbGripperScrewersDragLeadBefore1Actuator;
QbGripperScrewerStoperActuator;

P10_GripperScrewer.QbGripperScrewer1Actuator;
P10_GripperScrewer.QbGripperScrewer2Actuator;
P10_GripperScrewer.QbGripperScrewer1CatchActuator;
P10_GripperScrewer.QbGripperScrewer2CatchActuator;

		
(*************************** 641 **************************************)
QABPneumatic641ValveCoils[1].0	:= P02_Dispencers.QbDispencer1SuckingValveActuator;			//Siłownik:	zawór ssący 1		
QABPneumatic641ValveCoils[1].1	;											                           	                
QABPneumatic641ValveCoils[1].2	:= P02_Dispencers.QbDispencer2SuckingValveActuator;  		//Siłownik:	zawór ssący 2	
QABPneumatic641ValveCoils[1].3	; 										                               	           
QABPneumatic641ValveCoils[1].4	:= P02_Dispencers.QbDispencer3SuckingValveActuator;			//Siłownik:	zawór ssący 3		
QABPneumatic641ValveCoils[1].5	;									                                   	          
QABPneumatic641ValveCoils[1].6	:= P02_Dispencers.QbDispencer4SuckingValveActuator;			//Siłownik:	zawór ssący 4		
QABPneumatic641ValveCoils[1].7	;								

QABPneumatic641ValveCoils[2].0	:=	P02_Dispencers.QbDispencer1DosingValveActuator;			//Siłownik: zawór tłoczący 1 
QABPneumatic641ValveCoils[2].1	:=	NOT P02_Dispencers.QbDispencer1DosingValveActuator;                        
QABPneumatic641ValveCoils[2].2	:=	P02_Dispencers.QbDispencer2DosingValveActuator;			//Siłownik: zawór tłoczący 2 
QABPneumatic641ValveCoils[2].3	:=	NOT P02_Dispencers.QbDispencer2DosingValveActuator;                         
QABPneumatic641ValveCoils[2].4	:=	P02_Dispencers.QbDispencer3DosingValveActuator;			//Siłownik: zawór tłoczący 3
QABPneumatic641ValveCoils[2].5	:=	NOT P02_Dispencers.QbDispencer3DosingValveActuator;	                         
QABPneumatic641ValveCoils[2].6	:=  P02_Dispencers.QbDispencer4DosingValveActuator;			//Siłownik: zawór tłoczący 4
QABPneumatic641ValveCoils[2].7	:=	NOT P02_Dispencers.QbDispencer4DosingValveActuator ;                 

QABPneumatic641ValveCoils[3].0	:= P02_Dispencers.QbDispencer1DropCatcherValveActuator;		//Siłownik:	tacka ociekowa 1    
QABPneumatic641ValveCoils[3].1	;	                                                                   	                   
QABPneumatic641ValveCoils[3].2	:= P02_Dispencers.QbDispencer2DropCatcherValveActuator;		//Siłownik:	tacka ociekowa 2   
QABPneumatic641ValveCoils[3].3	;			                                                           	                         
QABPneumatic641ValveCoils[3].4	:= P02_Dispencers.QbDispencer3DropCatcherValveActuator;		//Siłownik:	tacka ociekowa 3	   
QABPneumatic641ValveCoils[3].5	;                                                                      	                 
QABPneumatic641ValveCoils[3].6	:= P02_Dispencers.QbDispencer4DropCatcherValveActuator; 	//Siłownik:	tacka ociekowa 4 
QABPneumatic641ValveCoils[3].7	;		                                                                                     

QABPneumatic641ValveCoils[4].0	:= P02_Dispencers.QbTank1Pressure	; //Nadciśnienie w zbiorniku masy  
QABPneumatic641ValveCoils[4].1	; //rezerwa
QABPneumatic641ValveCoils[4].2	:= NOT P02_Dispencers.QbDispencersCatch2Actuator;  
QABPneumatic641ValveCoils[4].3	:= NOT P02_Dispencers.QbDispencersCatch1Actuator;  
QABPneumatic641ValveCoils[4].4	:= NOT P02_Dispencers.QbDispencersCatch4Actuator;  
QABPneumatic641ValveCoils[4].5	:= NOT P02_Dispencers.QbDispencersCatch3Actuator;  
QABPneumatic641ValveCoils[4].6	;     
QABPneumatic641ValveCoils[4].7	;		    
                                
QABPneumatic641ValveCoils[5].0	:=  P02_Dispencers.QbDispencersCatch2Actuator;			//Siłownik: centrowanie szyjki 1	  
QABPneumatic641ValveCoils[5].1	:=  P02_Dispencers.QbDispencersCatch1Actuator;                                        
QABPneumatic641ValveCoils[5].2	:=  P02_Dispencers.QbDispencersCatch4Actuator; 				  
QABPneumatic641ValveCoils[5].3	:=  P02_Dispencers.QbDispencersCatch3Actuator;                  
QABPneumatic641ValveCoils[5].4	;				 
QABPneumatic641ValveCoils[5].5	;                   
QABPneumatic641ValveCoils[5].6	;					  
QABPneumatic641ValveCoils[5].7	; 

QABPneumatic641ValveCoils[6].0	;
QABPneumatic641ValveCoils[6].1	;
QABPneumatic641ValveCoils[6].2	;
QABPneumatic641ValveCoils[6].3	;
QABPneumatic641ValveCoils[6].4	;
QABPneumatic641ValveCoils[6].5	;
QABPneumatic641ValveCoils[6].6	;
QABPneumatic641ValveCoils[6].7	;

(***************************Koniec 641 **************************************)

(*************************** 642 **************************************)
QABPneumatic642ValveCoils[1].0	:= NOT p01_twophasesbarriers.QbBarrierBetweenDispencerActuator;
QABPneumatic642ValveCoils[1].1	:= 	   p01_twophasesbarriers.QbBarrierBetweenDispencerActuator; 
QABPneumatic642ValveCoils[1].2	:= NOT P01_TwoPhasesBarriers.QbBarrierBetweenWeightActuator;
QABPneumatic642ValveCoils[1].3	:=  P01_TwoPhasesBarriers.QbBarrierBetweenWeightActuator;
QABPneumatic642ValveCoils[1].4	:=     P02_Dispencers.QbDispencersDragLeftDragActuator;	
QABPneumatic642ValveCoils[1].5	:= NOT P02_Dispencers.QbDispencersDragLeftDragActuator;  
QABPneumatic642ValveCoils[1].6	:=     P02_Dispencers.QbDispencersDragRightDragActuator;		      
QABPneumatic642ValveCoils[1].7	:= NOT P02_Dispencers.QbDispencersDragRightDragActuator;		   		
                                        
QABPneumatic642ValveCoils[2].0	:=	   P02_Dispencers.QbDispencersDragLeftLeadBefore1Actuator;			  
QABPneumatic642ValveCoils[2].1	:= NOT P02_Dispencers.QbDispencersDragLeftLeadBefore1Actuator;  	            		
QABPneumatic642ValveCoils[2].2	:=	   P02_Dispencers.QbDispencersDragRightLeadBefore1Actuator;	
QABPneumatic642ValveCoils[2].3	:= NOT P02_Dispencers.QbDispencersDragRightLeadBefore1Actuator; 
QABPneumatic642ValveCoils[2].4	:=     P01_Gates.QbGate0BeforeDispencersActuator; 	//szlaban przed dozownikami wcześniejszy
QABPneumatic642ValveCoils[2].5	:= NOT P01_Gates.QbGate0BeforeDispencersActuator;  	
QABPneumatic642ValveCoils[2].6	:=		P01_Gates.QbGate0BeforeDispencersActuator;   ////szlaban przed dozownikami późniejszy              
QABPneumatic642ValveCoils[2].7	:=  NOT P01_Gates.QbGate0BeforeDispencersActuator;	           		
                                       
QABPneumatic642ValveCoils[3].0	:=   p01_gates.QbBottleTransferGate1Actuator;              
QABPneumatic642ValveCoils[3].1	:=  NOT p01_gates.QbBottleTransferGate1Actuator; 			
QABPneumatic642ValveCoils[3].2	:=   QbBlowAfterGripperScrewer;                 
QABPneumatic642ValveCoils[3].3	:=     P02_Dispencers.QbDispencerDropCatcherSuck;    
QABPneumatic642ValveCoils[3].4	;
QABPneumatic642ValveCoils[3].5	;
QABPneumatic642ValveCoils[3].6	;
QABPneumatic642ValveCoils[3].7	;
 
QABPneumatic642ValveCoils[4].0		; 
QABPneumatic642ValveCoils[4].1		; 
QABPneumatic642ValveCoils[4].2		; 
QABPneumatic642ValveCoils[4].3		; 
QABPneumatic642ValveCoils[4].4		; 
QABPneumatic642ValveCoils[4].5		; 
QABPneumatic642ValveCoils[4].6		; 
QABPneumatic642ValveCoils[4].7		;
 
QABPneumatic642ValveCoils[5].0		; 
QABPneumatic642ValveCoils[5].1		; 
QABPneumatic642ValveCoils[5].2		; 
QABPneumatic642ValveCoils[5].3		; 
QABPneumatic642ValveCoils[5].4		; 
QABPneumatic642ValveCoils[5].5		; 
QABPneumatic642ValveCoils[5].6		; 
QABPneumatic642ValveCoils[5].7		; 
(***************************Koniec 642 **************************************)

(*************************** 643 **************************************)
QABPneumatic643ValveCoils[1].0		:=	P05_Weight.QbWeight1Actuator;//QbWeight1ActuatorUp;			     :=  
QABPneumatic643ValveCoils[1].1		:=	NOT P05_Weight.QbWeight1Actuator;//QbWeight1ActuatorDown;        :=  
QABPneumatic643ValveCoils[1].2		:= 	P05_Weight.QbWeight2Actuator;//QbWeight2ActuatorUp; 		     :=  
QABPneumatic643ValveCoils[1].3		:= 	NOT P05_Weight.QbWeight2Actuator;//QbWeight2ActuatorDown;        := 
QABPneumatic643ValveCoils[1].4		:= 	P05_Weight.QbWeight3Actuator;//QbWeight3ActuatorUp; 		     := 
QABPneumatic643ValveCoils[1].5		:=  NOT P05_Weight.QbWeight3Actuator;//QbWeight3ActuatorDown;        := 
QABPneumatic643ValveCoils[1].6		:= 	P05_Weight.QbWeight4Actuator;//QbWeight4ActuatorUp;		         :=  
QABPneumatic643ValveCoils[1].7		:=  NOT P05_Weight.QbWeight4Actuator;//QbWeight4ActuatorDown;        :=  
                                                                                                         
QABPneumatic643ValveCoils[2].0		:=  P05_Weight.QbWeight5Actuator; 			                                       
QABPneumatic643ValveCoils[2].1		:=  NOT P05_Weight.QbWeight5Actuator;  			                                          
QABPneumatic643ValveCoils[2].2		:=  P05_Weight.QbWeight6Actuator; 		                                       
QABPneumatic643ValveCoils[2].3		:=  NOT P05_Weight.QbWeight6Actuator; 		                                          
QABPneumatic643ValveCoils[2].4		:= P01_Gates.QbGateBeforeWeight14Actuator;						                                                           
QABPneumatic643ValveCoils[2].5		:= NOT P01_Gates.QbGateBeforeWeight14Actuator;                                                               
QABPneumatic643ValveCoils[2].6		:= P01_gates.QbGateBeforeWeight56Actuator;						                                                           
QABPneumatic643ValveCoils[2].7		:= NOT P01_gates.QbGateBeforeWeight56Actuator;				                                                  
                                                                                                    
QABPneumatic643ValveCoils[3].0		:= P02_Dispencers.QbDispencersDragLeftLeadAfter1Actuator;		                                                         
QABPneumatic643ValveCoils[3].1		:= NOT P02_Dispencers.QbDispencersDragLeftLeadAfter1Actuator;	                                                           
QABPneumatic643ValveCoils[3].2		:= P02_Dispencers.QbDispencersDragrightLeadAfter1Actuator;		
QABPneumatic643ValveCoils[3].3		:= NOT P02_Dispencers.QbDispencersDragrightLeadAfter1Actuator;	
QABPneumatic643ValveCoils[3].4		; 
QABPneumatic643ValveCoils[3].5		; 
QABPneumatic643ValveCoils[3].6		; 
QABPneumatic643ValveCoils[3].7		;

QABPneumatic643ValveCoils[4].0		; 
QABPneumatic643ValveCoils[4].1		; 
QABPneumatic643ValveCoils[4].2		; 
QABPneumatic643ValveCoils[4].3		; 
QABPneumatic643ValveCoils[4].4		; 
QABPneumatic643ValveCoils[4].5		; 
QABPneumatic643ValveCoils[4].6		; 
QABPneumatic643ValveCoils[4].7		;
 
QABPneumatic643ValveCoils[5].0		; 
QABPneumatic643ValveCoils[5].1		; 
QABPneumatic643ValveCoils[5].2		; 
QABPneumatic643ValveCoils[5].3		; 
QABPneumatic643ValveCoils[5].4		; 
QABPneumatic643ValveCoils[5].5		; 
QABPneumatic643ValveCoils[5].6		; 
QABPneumatic643ValveCoils[5].7		; 
(***************************Koniec 643 **************************************)

(*************************** 644 **************************************)
QABPneumatic644ValveCoils[1].0		:=	P01_Gates.QbLidFeederBarrierActuator;
QABPneumatic644ValveCoils[1].1		:= NOT P01_Gates.QbLidFeederBarrierActuator;
QABPneumatic644ValveCoils[1].2		:= P06_WickFeeder.QbFormPositioning;
QABPneumatic644ValveCoils[1].3		:=FALSE;
QABPneumatic644ValveCoils[1].4		:= P06_WickFeeder.QbWickFeederDragLeadBefore1Actuator;  			
QABPneumatic644ValveCoils[1].5		:= NOT P06_WickFeeder.QbWickFeederDragLeadBefore1Actuator;  									
QABPneumatic644ValveCoils[1].6		:= P06_WickFeeder.QbWickFeederDragActuator;	                  
QABPneumatic644ValveCoils[1].7		:= NOT P06_WickFeeder.QbWickFeederDragActuator;	 	
                                            	
QABPneumatic644ValveCoils[2].0		:= P06_LidSealer.QbLidSealerDragLeadBefore1Actuator;	
QABPneumatic644ValveCoils[2].1		:= NOT P06_LidSealer.QbLidSealerDragLeadBefore1Actuator;		
QABPneumatic644ValveCoils[2].2		:=P06_LidSealer.QbLidSealerDragActuator;
QABPneumatic644ValveCoils[2].3		:= NOT P06_LidSealer.QbLidSealerDragActuator;
QABPneumatic644ValveCoils[2].4		:= P10_GripperScrewer.QbGripperScrewersDragLeadBefore1Actuator; 	  
QABPneumatic644ValveCoils[2].5		:= NOT P10_GripperScrewer.QbGripperScrewersDragLeadBefore1Actuator; 
QABPneumatic644ValveCoils[2].6		:= P10_GripperScrewer.QbGripperScrewersDragActuator;		 
QABPneumatic644ValveCoils[2].7		:= NOT P10_GripperScrewer.QbGripperScrewersDragActuator; 

QABPneumatic644ValveCoils[3].0		; //rezerwa
QABPneumatic644ValveCoils[3].1		; //rezerwa
QABPneumatic644ValveCoils[3].2		; //rezerwa
QABPneumatic644ValveCoils[3].3		; //rezerwa
QABPneumatic644ValveCoils[3].4		:= QbGripperScrewerAcceleratorActuator;
QABPneumatic644ValveCoils[3].5		:=FALSE;
QABPneumatic644ValveCoils[3].6		:= QbGripperScrewerStoperActuator;
QABPneumatic644ValveCoils[3].7		:=FALSE;
 
QABPneumatic644ValveCoils[4].0		:=P06_LidSealer.QbLidSealerStoperActuatorOn;
QABPneumatic644ValveCoils[4].1		:=FALSE; 
QABPneumatic644ValveCoils[4].2		; 
QABPneumatic644ValveCoils[4].3		; 
QABPneumatic644ValveCoils[4].4		; 
QABPneumatic644ValveCoils[4].5		; 
QABPneumatic644ValveCoils[4].6		; 
QABPneumatic644ValveCoils[4].7		;
 
QABPneumatic644ValveCoils[5].0		; 
QABPneumatic644ValveCoils[5].1		; 
QABPneumatic644ValveCoils[5].2		; 
QABPneumatic644ValveCoils[5].3		; 
QABPneumatic644ValveCoils[5].4		; 
QABPneumatic644ValveCoils[5].5		; 
QABPneumatic644ValveCoils[5].6		; 
QABPneumatic644ValveCoils[5].7		; 
(***************************Koniec 644 **************************************)

(*************************** 645 **************************************)
QABPneumatic645ValveCoils[1].0		:= P10_GripperScrewer.QbGripperScrewer2Actuator; 		
QABPneumatic645ValveCoils[1].1		:= P10_GripperScrewer.QbGripperScrewer1Actuator;		
QABPneumatic645ValveCoils[1].2		:= P10_GripperScrewer.QbGripperScrewer1CatchActuator;
QABPneumatic645ValveCoils[1].3		:= FALSE;                                            
QABPneumatic645ValveCoils[1].4		:= P10_GripperScrewer.QbGripperScrewer2CatchActuator;
QABPneumatic645ValveCoils[1].5		:= FALSE;                                            
QABPneumatic645ValveCoils[1].6		; 
QABPneumatic645ValveCoils[1].7		;
              
QABPneumatic645ValveCoils[2].0		; 
QABPneumatic645ValveCoils[2].1		; 
QABPneumatic645ValveCoils[2].2		; 
QABPneumatic645ValveCoils[2].3		; 
QABPneumatic645ValveCoils[2].4		; 
QABPneumatic645ValveCoils[2].5		; 
QABPneumatic645ValveCoils[2].6		; 
QABPneumatic645ValveCoils[2].7		;
(***************************Koniec 645 **************************************)

(*************************** 646 **************************************)
//Platynki
(*QABPneumatic646ValveCoils[1].0		:= P06_LidFeeder.QbLidFeeder2_FeederActuator1	;	//pobieranie i ruch w dół 						
QABPneumatic646ValveCoils[1].1		:= NOT P06_LidFeeder.QbLidFeeder2_FeederActuator1;    //pobieranie i ruch w dół                        
QABPneumatic646ValveCoils[1].2		:= P06_LidFeeder.QbLidFeeder2_FeederActuator2;		//wbicie wkładki       
QABPneumatic646ValveCoils[1].3		:= NOT P06_LidFeeder.QbLidFeeder2_FeederActuator2; 	//wbicie wkładki         
QABPneumatic646ValveCoils[1].4		:= P06_LidFeeder.QbLidFeeder_FeederActuator1	;	    //pobieranie wkładki 2                          
QABPneumatic646ValveCoils[1].5		:= NOT P06_LidFeeder.QbLidFeeder_FeederActuator1;  //pobieranie wkładki 2                              
QABPneumatic646ValveCoils[1].6		:= P06_LidFeeder.QbLidFeeder_FeederActuator2;		    //odkładanie wkładki 2                          
QABPneumatic646ValveCoils[1].7		:= NOT P06_LidFeeder.QbLidFeeder_FeederActuator2;  //odkładanie wkładki 2                              
                                                                                                
QABPneumatic646ValveCoils[2].0		;                                                          
QABPneumatic646ValveCoils[2].1		;                                                          
QABPneumatic646ValveCoils[2].2		;                                                          
QABPneumatic646ValveCoils[2].3		;                                                           
QABPneumatic646ValveCoils[2].4		;                                                           
QABPneumatic646ValveCoils[2].5		; 
QABPneumatic646ValveCoils[2].6		; 
QABPneumatic646ValveCoils[2].7		;
 
QABPneumatic646ValveCoils[3].0		:= P06_LidFeeder.QbLidFeeder_SuckerActuator ;
QABPneumatic646ValveCoils[3].1		:= P06_LidFeeder.QbLidFeeder2_SuckerActuator  ;*)
//Knoty
QABPneumatic646ValveCoils[1].0		:= NOT P06_WickFeeder.QbStopper1;	// u góry			           
QABPneumatic646ValveCoils[1].1		:= NOT P06_WickFeeder.QbStopper2;              
QABPneumatic646ValveCoils[1].2		:= P06_WickFeeder.QbSeparator1;			            
QABPneumatic646ValveCoils[1].3		:= P06_WickFeeder.QbSeparator2	;		         
QABPneumatic646ValveCoils[1].4		:= P06_WickFeeder.QbSleve1SeparatorActOut	;            
QABPneumatic646ValveCoils[1].5		:= P06_WickFeeder.QbSleve1SeparatorActIn	;                  
QABPneumatic646ValveCoils[1].6		:= P06_WickFeeder.QbSleve2SeparatorActOut	;                  
QABPneumatic646ValveCoils[1].7		:= P06_WickFeeder.QbSleve2SeparatorActIn	;                                                                 	           
QABPneumatic646ValveCoils[2].0		:=	P06_WickFeeder.QbHammer1;	            
QABPneumatic646ValveCoils[2].1		:=	NOT P06_WickFeeder.QbHammer1;	      ;     
QABPneumatic646ValveCoils[2].2		:= 	P06_WickFeeder.QbHammer2			      ; 
QABPneumatic646ValveCoils[2].3		:=  NOT P06_WickFeeder.QbHammer2			 		  ;
QABPneumatic646ValveCoils[2].4		:=  P06_WickFeeder.QbBlow1	;		
QABPneumatic646ValveCoils[2].5		:= P06_WickFeeder.QbSleeveBlow;			
QABPneumatic646ValveCoils[2].6		;
QABPneumatic646ValveCoils[2].7		;
                                    
QABPneumatic646ValveCoils[3].0		;
QABPneumatic646ValveCoils[3].1		;
(***************************Koniec 646 **************************************)

(*************************** 647**************************************)
// Wyspa 647 - podajnik opakowań
QABPneumatic647ValveCoils[1].0 := P08_CapSorter.QbCapSorterDragActuator;     //[710, 5/3, wysunięcie wideł]
QABPneumatic647ValveCoils[1].1 := NOT P08_CapSorter.QbCapSorterDragActuator;					
QABPneumatic647ValveCoils[1].2 := P08_CapSorter.QbCapSorterDragLeadBefore1Actuator;    //[720, 5/3 , wysunięcie prowaadzenie ]
QABPneumatic647ValveCoils[1].3 := NOT P08_CapSorter.QbCapSorterDragLeadBefore1Actuator;
QABPneumatic647ValveCoils[1].4 := P08_CapSorter.QbCapSorterStoperActuator;   //[730, 5/2, wysunięcie amortyzatora]
QABPneumatic647ValveCoils[1].5;
QABPneumatic647ValveCoils[1].6 := P08_CapSorter.QbCapSorterDragLeadAfter1Actuator;
QABPneumatic647ValveCoils[1].7 := NOT P08_CapSorter.QbCapSorterDragLeadAfter1Actuator;
QABPneumatic647ValveCoils[2].0;
QABPneumatic647ValveCoils[2].1 := QbBlowBeforeGripperScrewer;//nie ma
QABPneumatic647ValveCoils[2].2 := QbGripperScrewerGateBeforeActuator; //nie ma
QABPneumatic647ValveCoils[2].3;
(*********************Koniec 647 **************************************)

(*************************** 641 **************************************)
QABPneumaticPI641ValveCoils[1].0	:= NOT P01_pucksInserter.QbPucksInserterHammer;
QABPneumaticPI641ValveCoils[1].1	:= P01_pucksInserter.QbPucksInserterHammer;					
QABPneumaticPI641ValveCoils[1].2	:= P01_pucksInserter.QbPucksInserterTray;
QABPneumaticPI641ValveCoils[1].3	:= NOT P01_pucksInserter.QbPucksInserterTray;
QABPneumaticPI641ValveCoils[1].4	:= NOT P01_pucksInserter.QbPucksInserterGate1;
QABPneumaticPI641ValveCoils[1].5	:=  P01_pucksInserter.QbPucksInserterGate1;
QABPneumaticPI641ValveCoils[1].6	:=  NOT P01_pucksInserter.QbPucksInserterGate2;
QABPneumaticPI641ValveCoils[1].7	:=  P01_pucksInserter.QbPucksInserterGate2;
QABPneumaticPI641ValveCoils[2].0 	:=  NOT P01_pucksInserter.QbPucksInserterFormGate;
QABPneumaticPI641ValveCoils[2].1	:=  P01_pucksInserter.QbPucksInserterFormGate;
QABPneumaticPI641ValveCoils[2].2	:=  NOT P01_pucksInserter.QbPucksInserterFormPositioning;
QABPneumaticPI641ValveCoils[2].3  :=  FALSE;//:= NOT P01_PucksInserter.QbPucksInserterPushTable_Gate;    //Vasyl 27.05 [670, 5/2 Szlabany stołu podającego]                    
QABPneumaticPI641ValveCoils[2].4	;//:= 	P01_PucksInserter.QbPucksInserterPushTable_Gate;	
QABPneumaticPI641ValveCoils[2].5;
QABPneumaticPI641ValveCoils[2].6	;//:= P01_PucksInserter.QbPucksInserterPushTable_Pushers; //Vasyl 04.08   [5/2 Popychacze stołu podającego]
QABPneumaticPI641ValveCoils[2].7;
(*********************Koniec 641 **************************************)
END_ACTION

ACTION aVTEM:
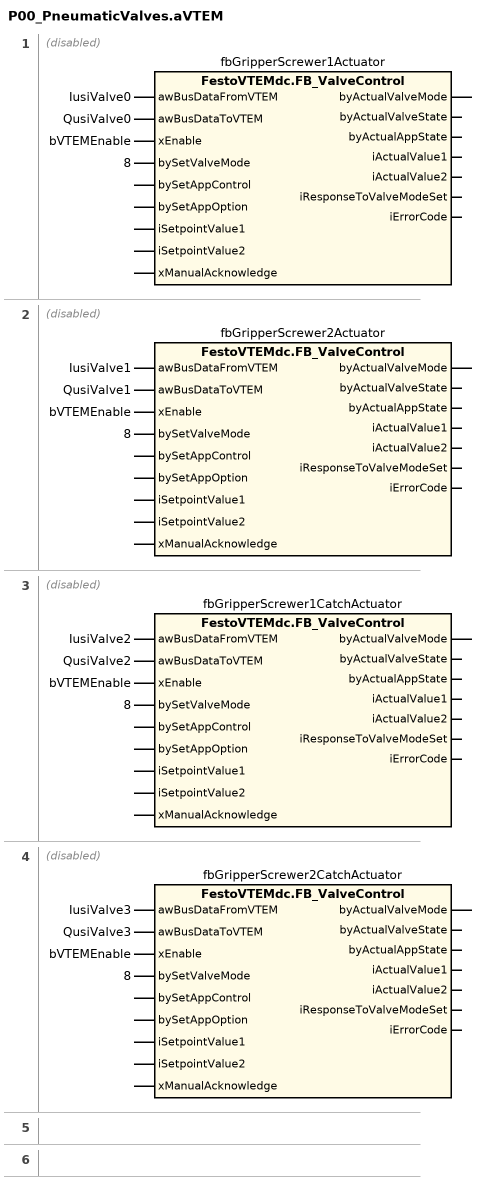
// NETWORK 1 (disabled)
// fbGripperScrewer1Actuator(
//     awBusDataFromVTEM := IusiValve0,
//     awBusDataToVTEM := QusiValve0,
//     xEnable := bVTEMEnable,
//     bySetValveMode := 8); // FestoVTEMdc.FB_ValveControl

// NETWORK 2 (disabled)
// fbGripperScrewer2Actuator(
//     awBusDataFromVTEM := IusiValve1,
//     awBusDataToVTEM := QusiValve1,
//     xEnable := bVTEMEnable,
//     bySetValveMode := 8); // FestoVTEMdc.FB_ValveControl

// NETWORK 3 (disabled)
// fbGripperScrewer1CatchActuator(
//     awBusDataFromVTEM := IusiValve2,
//     awBusDataToVTEM := QusiValve2,
//     xEnable := bVTEMEnable,
//     bySetValveMode := 8); // FestoVTEMdc.FB_ValveControl

// NETWORK 4 (disabled)
// fbGripperScrewer2CatchActuator(
//     awBusDataFromVTEM := IusiValve3,
//     awBusDataToVTEM := QusiValve3,
//     xEnable := bVTEMEnable,
//     bySetValveMode := 8); // FestoVTEMdc.FB_ValveControl

// NETWORK 5

// NETWORK 6
END_ACTION

ACTION aVTEMSignals:
// Wszystkie od 1 do 8 bar
(*
(********VTEM 0********)
(***     F[N]=p[bar]*14,8[N/bar] ************) // od 1,5kg do 12kg
IF lrGripperScrewerPressure = 0 					THEN	lrGripperScrewerPressure := 2; 						END_IF;
IF lrGripperScrewerPressureExhaustLevel < 10	THEN	lrGripperScrewerPressureExhaustLevel := 10;		END_IF;
fbGripperScrewer1Actuator.iSetpointValue2 := (**Smbar Setpoint sir supply pressure during travel**)
ABS(LREAL_TO_INT(((lrGripperScrewerPressure*10)/14.8)*1000));
IF fbGripperScrewer1Actuator.iSetpointValue2 >8000 THEN
	fbGripperScrewer1Actuator.iSetpointValue2 := 8000;
END_IF
IF fbGripperScrewer1Actuator.iSetpointValue2 >8000 THEN
	fbGripperScrewer1Actuator.iSetpointValue2 := 8000;
END_IF
IF P10_GripperScrewer.QbGripperScrewer1Actuator THEN(**Włączanie zaworu**)
	fbGripperScrewer1Actuator.bySetAppControl	:= 2;
	fbGripperScrewer1Actuator.iSetpointValue1	:= LREAL_TO_INT(lrGripperScrewerPressureExhaustLevel*100);//10000;(**Setpoint opening degree axhaust air flow control**)
ELSE
	fbGripperScrewer1Actuator.bySetAppControl	:= 3;
	fbGripperScrewer1Actuator.iSetpointValue1	:= 10000;(**Setpoint opening degree axhaust air flow control**)
END_IF	
IF fbGripperScrewer1Actuator.iResponseToValveModeSet = 1037 (*Acknoledge_needed*) THEN
	fbGripperScrewer1Actuator.xManualAcknowledge := TRUE;	ELSE
	fbGripperScrewer1Actuator.xManualAcknowledge := FALSE;	END_IF
	
	
(********VTEM 1********)
(***     F[N]=p[bar]*14,8[N/bar] ************) // od 1,5kg do 12kg
IF lrGripperScrewerPressure = 0 					THEN	lrGripperScrewerPressure := 2; 						END_IF;
IF lrGripperScrewerPressureExhaustLevel < 10	THEN	lrGripperScrewerPressureExhaustLevel := 10;		END_IF;
fbGripperScrewer2Actuator.iSetpointValue2 := (**Smbar Setpoint sir supply pressure during travel**)
ABS(LREAL_TO_INT(((lrGripperScrewerPressure*10)/14.8)*1000));
IF fbGripperScrewer2Actuator.iSetpointValue2 >8000 THEN
	fbGripperScrewer2Actuator.iSetpointValue2 := 8000;
END_IF
IF fbGripperScrewer2Actuator.iSetpointValue2 >8000 THEN
	fbGripperScrewer2Actuator.iSetpointValue2 := 8000;
END_IF
IF P10_GripperScrewer.QbGripperScrewer2Actuator THEN(**Włączanie zaworu**)
	fbGripperScrewer2Actuator.bySetAppControl	:= 2;
	fbGripperScrewer2Actuator.iSetpointValue1	:= LREAL_TO_INT(lrGripperScrewerPressureExhaustLevel*100);(**Setpoint opening degree axhaust air flow control**)
ELSE
	fbGripperScrewer2Actuator.bySetAppControl	:= 3;
	fbGripperScrewer2Actuator.iSetpointValue1	:= 10000;(**Setpoint opening degree axhaust air flow control**)
END_IF	
IF fbGripperScrewer2Actuator.iResponseToValveModeSet = 1037 (*Acknoledge_needed*) THEN
	fbGripperScrewer2Actuator.xManualAcknowledge := TRUE;	ELSE
	fbGripperScrewer2Actuator.xManualAcknowledge := FALSE;	END_IF
	
	
(********VTEM 2********)
IF lrGripperScrewerPressure = 0 					THEN	lrGripperScrewerPressure := 3; 						END_IF;
IF (lrGripperScrewerCatchPressureExhaustLevel < 10)	THEN	lrGripperScrewerCatchPressureExhaustLevel := 10;		END_IF; // bylo <1000
fbGripperScrewer1CatchActuator.iSetpointValue2 := (**Smbar Setpoint sir supply pressure during travel**)
ABS(LREAL_TO_INT(((lrGripperScrewerPressure*10)/26.2)*1000));
IF fbGripperScrewer1CatchActuator.iSetpointValue2 >8000 THEN
	fbGripperScrewer1CatchActuator.iSetpointValue2 := 8000;
END_IF
IF P10_GripperScrewer.QbGripperScrewer1CatchActuator THEN(**Włączanie zaworu**)
	fbGripperScrewer1CatchActuator.bySetAppControl	:= 1;
	fbGripperScrewer1CatchActuator.iSetpointValue1	:= LREAL_TO_INT((lrGripperScrewerCatchPressureExhaustLevel*15.5)-55);(**Setpoint opening degree axhaust air flow control**)
ELSE
	fbGripperScrewer1CatchActuator.bySetAppControl	:= 2;
	fbGripperScrewer1CatchActuator.iSetpointValue1	:= 10000;(**Setpoint opening degree axhaust air flow control**)
END_IF
IF fbGripperScrewer1CatchActuator.iResponseToValveModeSet = 1037 (*Acknoledge_needed*) THEN
	fbGripperScrewer1CatchActuator.xManualAcknowledge := TRUE;	ELSE
	fbGripperScrewer1CatchActuator.xManualAcknowledge := FALSE;	END_IF	
		
	
(********VTEM 3********)
IF lrGripperScrewerPressure = 0 					THEN	lrGripperScrewerPressure := 3; 						END_IF;
IF ((lrGripperScrewerCatchPressureExhaustLevel) < 10)	THEN	lrGripperScrewerCatchPressureExhaustLevel := 10;		END_IF; // było <1000 i 100000

fbGripperScrewer2CatchActuator.iSetpointValue2 := (**Smbar Setpoint sir supply pressure during travel**)
ABS(LREAL_TO_INT(((lrGripperScrewerPressure*10)/26.2)*1000));
IF fbGripperScrewer2CatchActuator.iSetpointValue2 >8000 THEN
	fbGripperScrewer2CatchActuator.iSetpointValue2 := 8000;
END_IF
IF P10_GripperScrewer.QbGripperScrewer2CatchActuator THEN(**Włączanie zaworu**)
	fbGripperScrewer2CatchActuator.bySetAppControl	:= 1;
	fbGripperScrewer2CatchActuator.iSetpointValue1	:= LREAL_TO_INT((lrGripperScrewerCatchPressureExhaustLevel*15.5)-55);(**Setpoint opening degree axhaust air flow control**)
ELSE
	fbGripperScrewer2CatchActuator.bySetAppControl	:= 2;
	fbGripperScrewer2CatchActuator.iSetpointValue1	:= 10000;(**Setpoint opening degree axhaust air flow control**)
END_IF
IF fbGripperScrewer2CatchActuator.iResponseToValveModeSet = 1037 (*Acknoledge_needed*) THEN
	fbGripperScrewer2CatchActuator.xManualAcknowledge := TRUE;	ELSE
	fbGripperScrewer2CatchActuator.xManualAcknowledge := FALSE;	END_IF	
			
	
*)
END_ACTION

END_PROGRAM

(* stored: Version 1.1.0.1, ProductVersion 3.1.4026.13, FileIdentifier 8218ebeeb92ae195bf7ec7d12e9843aa282c3100, FileSignature 3de39c3480f1f1431f9222abcbaa96233e2bd5d3bf68d3db8943c628d47b73b118e3f0996f984ddc09ee205a06260789f5987581d11ba5973cb3a3639f56541480db0b7c968c31f2cf0909f3e8a32f528bc09974b83da1c94479454fd3d318b461e4cb42106a431b2c245cad64206441eb8055efcd86d1163e752e143c4affd8546f7084b5eeb08003da42388dcb85800f9f31e84515ba2b0c430466ac5420a657af11040f42ac8388ee6732656848a2070d8183c04e3ab79057407d11ff9c4047afc8365fc3bf0709dab516b881d21732bb6408b29ae464baf0b2e786264410a19ad3ae34dbb0bafff87c9c7158b299ca62aec08ca31b0ea33c0ffd2215de9a
   POU P00_PneumaticValves: Id {ee66e38d-fe20-4ed1-a6a8-8b7178c0f4b0}, SpecialFunc None
   Action aAnalogueInput: Id {a8f125df-6e95-4681-8771-606ae0865b15}
   Action aDigitalInput: Id {6775fd0f-6e49-4e73-a900-876f1e5f71c1}
   Action aPressureRegulator: Id {d2f8e272-44ff-4f57-9dc7-018d20b4cc14}
   Action aValveCoil: Id {6eea7603-0c5d-469c-a72c-ddd9e83354d1}
   Action aVTEM: Id {53c485ad-497f-428a-b9a9-4f2e50c67e0a}
   Action aVTEMSignals: Id {b40f8d87-5947-4185-8bde-4a7782a35bb6} *)
